(* CoDeSys 2.3.9.47 project: wtp_13_05_16.pro *)
(* Libraries: TcBase.lib 14.5.09 12:14:08, TcSystem.lib 21.1.15 10:22:54, TcBaseMath.lib 27.7.04 12:07:56, TcMath.lib 23.9.04 15:15:30, TcMC2.lib 19.10.15 14:49:44, STANDARD.LIB 5.6.98 12:03:02 *)

(* Task configuration *)
TASK Standard (PRIORITY := 0, INTERVAL := T#10ms);
	MAIN
END_TASK

(* POU MAIN, ST *)
PROGRAM MAIN
VAR
	test : rus_pump_mixer_start;
	test_stop : rus_pump_mixer_stop;
	a : st_rus_pump_mixer_DNA;
	test3:rus_inlet_eq_sbr;
	b: st_rus_inlet_eq_sbr_DNA;
END_VAR
test(a:=a);
test_stop(a:=a);
test3(a:=a,b:=b);
END_PROGRAM

(* POU rus_pump_mixer_start, ST *)
FUNCTION_BLOCK rus_pump_mixer_start
VAR_INPUT
END_VAR
VAR_OUTPUT
END_VAR
VAR
	startPumpMixerDelayTimer: TON;
END_VAR
VAR_IN_OUT
	a : st_rus_pump_mixer_DNA;
END_VAR
CASE a.startSeq OF
0:
	IF a.bStartPumpMixer THEN
		a.startSeq := 100;
		a.bBusy := TRUE;
		a.bDone := FALSE;

	(*
		a.bErrorDuty := FALSE;
		a.bErrorStandby := FALSE;
		a.bErrorCriticalStart := FALSE;
		a.bErrorIsInManualDuty := FALSE;
		a.bErrorIsInManualStandby := FALSE;
	

	a.bErrorOverloadDuty:= FALSE;
	a.bErrorIncompleteDuty:= FALSE;
	a.bErrorStartStopStatDuty:= FALSE;
	a.bErrorOverloadStandby:= FALSE;
	a.bErrorIncompleteStandby:= FALSE;
	a.bErrorStartStopStatStandby:= FALSE;
	*)

	a.bCmdStartDuty := FALSE;
	a.bCmdStartStandby := FALSE;
	END_IF
100:
	IF a.bRemoteDuty THEN
		a.startSeq := 200;
	ELSE
		a.startSeq := 9000;
		a.bErrorIsInManualDuty := TRUE;
	END_IF
200:
	a.bCmdStartDuty := TRUE;
	startPumpMixerDelayTimer(IN:=TRUE , PT:=a.startPumpMixerDelay);
	IF startPumpMixerDelayTimer.Q THEN
		startPumpMixerDelayTimer(IN:=FALSE);
		a.startSeq := 230;
	END_IF
230:
	a.bErrorDuty := TRUE;
	a.startSeq := 5000;
	IF a.bOverloadDuty THEN
		a.bErrorOverloadDuty := TRUE;
	ELSIF a.bIncompleteDuty THEN
		a.bErrorIncompleteDuty := TRUE;
	ELSIF NOT  a.bStartStopStatDuty THEN
		a.bErrorStartStopStatDuty := TRUE;
	ELSE
		a.bErrorDuty := FALSE;
		a.startSeq := 500;
	END_IF
500:
	a.bCmdStartStandby := FALSE;
	a.bDone := TRUE;
	a.startSeq := 9000;
5000:
	IF a.bRemoteStandby THEN
		a.startSeq := 5100;
	ELSE
		a.bErrorisInManualStandby := TRUE;
		a.startSeq:= 9000;
	END_IF
5100:
	a.bCmdStartStandby := TRUE;
	a.bCmdStartDuty := FALSE;
	startPumpMixerDelayTimer(IN:=TRUE, PT:=a.startPumpMixerDelay);
	IF startPumpMixerDelayTimer.Q THEN
		startPumpMixerDelayTimer(IN:=FALSE);
		a.startSeq := 5200;
	END_IF
5200:
	a.bErrorStandby := TRUE;
	a.startSeq := 5150;
	IF a.bOverloadStandby THEN
		a.bErrorOverloadStandby := TRUE;
	ELSIF a.bIncompleteStandby THEN
		a.bErrorIncompleteStandby := TRUE;
	ELSIF NOT  a.bStartStopStatStandby THEN
		a.bErrorStartStopStatStandby := TRUE;
	ELSE
	a.bErrorStandby := FALSE;
	a.bDone:=TRUE;
		a.startSeq := 9000;
	END_IF
5150:
	IF a.bRemoteDuty THEN
		a.startSeq := 5250;
	ELSE
		a.startSeq := 9000;
		a.bErrorIsInManualDuty := TRUE;
	END_IF
5250:
	a.bCmdStartDuty := TRUE;
	startPumpMixerDelayTimer(IN:=TRUE , PT:=a.startPumpMixerDelay);
	IF startPumpMixerDelayTimer.Q THEN
		startPumpMixerDelayTimer(IN:=FALSE);
		a.startSeq := 5300;
	END_IF
5300:
	a.bErrorCriticalStart :=TRUE;
	a.startSeq := 9000;
	IF a.bOverloadDuty THEN
		a.bErrorOverloadDuty := TRUE;
	ELSIF a.bIncompleteDuty THEN
		a.bErrorIncompleteDuty := TRUE;
	ELSIF NOT  a.bStartStopStatDuty THEN
		a.bErrorStartStopStatDuty := TRUE;
	ELSE
		a.bErrorCriticalStart :=FALSE;
		a.bErrorDuty := FALSE;
		a.startSeq := 5400;
	END_IF
5400:
	a.bCmdStartStandby := FALSE;
	a.startSeq:= 9000;
	a.bDone := TRUE;
9000:
	a.bBusy := FALSE;
	IF NOT a.bStartPumpMixer OR a.bStopPumpMixer THEN
	a.bDone := FALSE;

	(*
	a.bErrorDuty := FALSE;
	a.bErrorStandby := FALSE;
	a.bErrorCriticalStart := FALSE;
	a.bErrorisInManualDuty := FALSE;
	a.bErrorIsInManualStandby := FALSE;
	*)
	
	a.startSeq:= 0;
	END_IF
END_CASE

IF a.bCLRErrorStartPumpMixer THEN
	a.bErrorDuty := FALSE;
	a.bErrorStandby := FALSE;
	a.bErrorCriticalStart := FALSE;
	a.bErrorIsInManualDuty := FALSE;
	a.bErrorIsInManualStandby := FALSE;

	a.bErrorOverloadDuty:= FALSE;
	a.bErrorIncompleteDuty:= FALSE;
	a.bErrorStartStopStatDuty:= FALSE;
	a.bErrorOverloadStandby:= FALSE;
	a.bErrorIncompleteStandby:= FALSE;
	a.bErrorStartStopStatStandby:= FALSE;
END_IF
END_FUNCTION_BLOCK

(* POU st_rus_pump_mixer_DNA, ST *)
FUNCTION_BLOCK st_rus_pump_mixer_DNA
VAR_INPUT
	bStartPumpMixer: BOOL;
	bStopPumpMixer : BOOL;

	bErrorOverloadDuty: BOOL;
	bErrorIncompleteDuty: BOOL;
	bErrorStartStopStatDuty: BOOL;

	bErrorOverloadStandby: BOOL;
	bErrorIncompleteStandby: BOOL;
	bErrorStartStopStatStandby: BOOL;

	bCmdStartDuty AT%Q*: BOOL;
	bCmdStartStandby AT%Q*: BOOL;

	bErrorIsInManualDuty : BOOL;
	bErrorIsInManualStandby : BOOL;
	bErrorDuty: BOOL;
	bErrorStandby: BOOL;

	bErrorCriticalStart: BOOL;
	bErrorCriticalStop:BOOL;

	bBusy:BOOL;
	bDone: BOOL;

	startSeq: INT;
	stopSeq:INT;

	bESTOP AT%Q* : BOOL;

	bCLRErrorStartPumpMixer : BOOL;
	bCLRErrorStopPumpMixer : BOOL;
END_VAR
VAR_OUTPUT


	bRemoteDuty AT%I*: BOOL;
	bRemoteStandby AT%I*: BOOL;

	bIncompleteDuty AT%I*: BOOL;
	bStartStopStatDuty AT%I*: BOOL;
	bOverloadDuty AT%I*: BOOL;


	bOverloadStandby AT%I*: BOOL;
	bIncompleteStandby AT%I*: BOOL;
	bStartStopStatStandby AT%I*: BOOL;

	startPumpMixerDelay: TIME := T#2s;

END_VAR
VAR
END_VAR
;
END_FUNCTION_BLOCK

(* POU rus_pump_mixer_stop, ST *)
FUNCTION_BLOCK rus_pump_mixer_stop
VAR_INPUT
END_VAR
VAR_OUTPUT
END_VAR
VAR

	timer_stop_duty : TON;
	timer_stop_standby :TON;
END_VAR
VAR_IN_OUT
	a : st_rus_pump_mixer_DNA;
END_VAR
CASE a.stopSeq OF
0:
 	IF a.bStopPumpMixer THEN
		a.stopSeq := 100;

		a.bBusy := TRUE;
	(*
		a.bErrorCriticalStop := FALSE;
		a.bESTOP := FALSE;
	*)
	END_IF
100:
	IF a.bRemoteDuty THEN
		a.bCmdStartDuty := FALSE;
	ELSE
		a.bErrorIsInManualDuty := TRUE;
	END_IF

	IF a.bRemoteStandby THEN
		a.bCmdStartStandby := FALSE;
	ELSE
		a.bErrorIsInManualStandby := TRUE;
	END_IF

	a.stopSeq := 300;
300:
	timer_stop_duty(IN:=TRUE,pt:=a.startPumpMixerDelay);
	IF timer_stop_duty.Q THEN
	timer_stop_duty(IN:=FALSE);
		IF a.bStartStopStatDuty  AND NOT a.bErrorIsInManualStandby THEN
			a.bESTOP := TRUE;
			a.bErrorCriticalStop := TRUE;
		END_IF
		IF a.bStartStopStatStandby  AND NOT a.bErrorIsInManualStandby THEN
			a.bESTOP := TRUE;
			a.bErrorCriticalStop := TRUE;
		END_IF
	a.stopSeq := 900;
	END_IF
900:
	a.bBusy := FALSE;
	IF  NOT a.bStopPumpMixer OR a.bStartPumpMixer THEN
		a.stopSeq := 0;
		(*
		a.bErrorCriticalStop := FALSE;
		a.bErrorIsInManualDuty := FALSE;
		a.bErrorIsInManualStandby := FALSE;
		*)
	END_IF
END_CASE

IF a.bCLRErrorStopPumpMixer THEN
	a.bErrorIsInManualDuty := FALSE;
	a.bErrorIsInManualStandby := FALSE;
	a.bESTOP := FALSE;
	a.bErrorCriticalStop := FALSE;
END_IF
END_FUNCTION_BLOCK

(* POU rus_inlet_eq_sbr, ST *)
FUNCTION_BLOCK rus_inlet_eq_sbr
VAR_INPUT
END_VAR
VAR_OUTPUT
END_VAR
VAR
END_VAR
VAR_IN_OUT
	a : st_rus_pump_mixer_DNA;
	b : st_rus_inlet_eq_sbr_DNA;
END_VAR
CASE b.eq_seq OF
0:
	b.eq_seq := 100;
100:
	IF b.bEQFloatSensorLO THEN
		b.eq_seq := 200;
	ELSE
		b.eq_seq := 600; (*stopping the pump*)
	END_IF
200:
	IF b.bEQFloatSensorOP THEN
		b.eq_seq := 300; (*evaluate condition b4 starting*)
	ELSE
		b.eq_seq := 500; (*stop pump*)
	END_IF
300:
	IF b.bEQFloatSensorHI THEN
		b.bErrorCritical_SEQ := TRUE;
		b.eq_seq := 350; (*evaluate condition b4 stopping*)
	ELSE
		b.eq_seq := 400; (*start pump*)
	END_IF
350:
	IF b.bSBRFloatSensor OR b.bStreamLineSensorOverflow THEN
		b.eq_seq := 500;(*stop pump*)
	ELSE
		b.eq_seq := 400; (*start pump*)
	END_IF
400:
	IF NOT (a.bCmdStartDuty OR a.bCmdStartStandby) THEN
		a.bStartPumpMixer :=TRUE;
	END_IF
		b.eq_seq := 450;
450:
	IF NOT a.bBusy THEN
		a.bStartPumpMixer :=FALSE;
		b.eq_seq := 900;
	END_IF
500:
	IF (a.bCmdStartDuty OR a.bCmdStartStandby) THEN
		a.bStopPumpMixer :=TRUE;
	END_IF
		b.eq_seq := 550;
550:
	IF NOT a.bBusy THEN
		a.bStopPumpMixer :=FALSE;
		b.eq_seq := 900;
	END_IF
600:
	IF (a.bStartStopStatDuty OR a.bStartStopStatStandby) THEN
		a.bStopPumpMixer :=TRUE;
	END_IF
		b.eq_seq := 650;
650:
	IF NOT a.bBusy THEN
		a.bStopPumpMixer :=FALSE;
		b.eq_seq := 700;
	END_IF
700:
	IF b.bEQFloatSensorDRY THEN
		b.bErrorWarning_SEQ:= TRUE;
	ELSE
		b.bErrorCritical_SEQ :=TRUE;
	END_IF
	b.eq_seq := 900;
900:
	(*return*)
	b.eq_seq := 0;
END_CASE

IF b.bCLRErrorSEQ THEN
b.bCLRErrorSEQ := FALSE;
b.bErrorCritical_SEQ := FALSE;
b.bErrorWarning_SEQ := FALSE;
a.bCLRErrorStartPumpMixer := TRUE;
a.bCLRErrorStopPumpMixer := TRUE;
ELSE
a.bCLRErrorStartPumpMixer := FALSE;
a.bCLRErrorStopPumpMixer := FALSE;
END_IF
END_FUNCTION_BLOCK

(* POU st_rus_inlet_eq_sbr_DNA, ST *)
FUNCTION_BLOCK st_rus_inlet_eq_sbr_DNA
VAR_INPUT
	eq_seq: INT;
	bCLRErrorSEQ: BOOL;
	bErrorWarning_SEQ: BOOL;
	bErrorCritical_SEQ: BOOL;
END_VAR
VAR_OUTPUT
	bEQFloatSensorLO AT%I*: BOOL;
	bEQFloatSensorOP AT%I*: BOOL;
	bEQFloatSensorHI AT%I*: BOOL;
	bEQFloatSensorDRY AT%I*: BOOL;

	bStreamLineSensorOverflow AT%I*: BOOL;
	bSBRFloatSensor AT%I*: BOOL;
END_VAR
VAR
END_VAR
;
END_FUNCTION_BLOCK

(* POU rus_mixer_eq_sbr, ST *)
PROGRAM rus_mixer_eq_sbr
VAR
END_VAR
;
END_PROGRAM
